PROGRAM P_Demo_PVOID_TO_BINSTR
VAR
    pTarget    : POINTER TO BYTE; // 测试用指针；演示中用 ADR(nProbe) 取实际地址
    nProbe     : BYTE := 16#5A; // 被指向的局部变量，用 ADR() 后地址作为 PVOID 输入
    sFormatted : STRING(255); // 主输出，在线 monitor 这一行看转换结果
END_VAR

// =============================================================================
// 场景：把 PVOID 指针 转为二进制 (base 2)定长字符串后用于 HMI 显示、日志或协议帧。
//       例：订单号、错误码、IO 状态位等场景需要"前补 0 到固定 6 位"。
// 价值：替代手写循环或 IEC 标准 STRING 转换 + 补零拼接，一行解决补零、保留全长、
//       空值（in=0 且 iPrecision=0 -> ''）三件事。
// 验证步骤：
//   1. 引用 Tc2_Utilities
//   2. 把本 PROGRAM 加进 PlcTask 任务调用列表
//   3. 编译 + 登录 + 运行
//   4. 在线 monitor sFormatted；改输入看输出变化
//      - 默认值, iPrecision = 6 -> 应是补零后的字符串
//      - 在线把 iPrecision 类参数换大（如改成 10）-> 字符串变长但前置 0 增多
//      - 把数值改 0、iPrecision 改 0 -> 返回 ''（验证空字符串特例）
// =============================================================================

pTarget := ADR(nProbe);  // 给指针赋实际地址，模拟运行时拿到一个内存地址
// 单行调用：得到二进制 (base 2)字符串
sFormatted := PVOID_TO_BINSTR(pTarget, 6);

END_PROGRAM

(* stored: Version 1.1.0.1, ProductVersion 3.1.4024.5
   POU P_Demo_PVOID_TO_BINSTR: Id {082a860d-0e81-5db5-a576-87bbc660bb24}, SpecialFunc None *)
